FUNCTION_BLOCK SoEReadProcess EXTENDS BaseProcess
  VAR_INPUT
    value1Byte : USINT;  (* Value that has been read, if noOfBytes is 1 *)
    value2Bytes : UINT;  (* Value that has been read, if noOfBytes is 2 *)
    value4Bytes : UDINT;  (* Value that has been read, if noOfBytes is 4 *)
    adsErrorId : UINT;  (* ADS error ID *)
    sercosErrorId : UINT;  (* Sercos error ID *)
    {attribute 'OPC.UA.DA' := '1'}
    set : SoEReadProcessArgs;  (* Arguments to be set, before writing do_request TRUE *)
  END_VAR
  VAR_OUTPUT
    {attribute 'OPC.UA.DA' := '1'}
    {attribute 'OPC.UA.DA.Access' := '1'}
    get : SoEReadProcessArgs;  (* Arguments in use by the process, if do_request was accepted *)
  END_VAR

            IF do_request THEN
    do_request_result := request(
    index := set.index,
    noOfBytes := set.noOfBytes);
    do_request := FALSE;
END_IF;
SUPER^();

          

{attribute 'TcRpcEnable' := '1'}
METHOD start
  VAR_INPUT
    index : UINT;  (* SDO Index *)
    noOfBytes : UDINT;  (* Number of bytes to be read *)
  END_VAR
                  THIS^.get.index := index;
THIS^.get.noOfBytes := noOfBytes;
THIS^.statuses.busyStatus( isBusy := TRUE );
THIS^.statuses.healthStatus( isGood := TRUE );

                
END_METHOD

{attribute 'TcRpcEnable' := '1'}
METHOD request : RequestResults
  VAR_INPUT
    index : UINT;  (* SDO Index *)
    noOfBytes : UDINT;  (* Number of bytes to be read *)
  END_VAR
                  IF THIS^.statuses.enabledStatus.enabled THEN
    request := RequestResults.ACCEPTED;
    THIS^.start(
        index := index,
        noOfBytes := noOfBytes);
ELSE
    request := RequestResults.REJECTED;
END_IF;

                
END_METHOD
END_FUNCTION_BLOCK

FUNCTION_BLOCK SoEWriteProcess EXTENDS BaseProcess
  VAR_INPUT
    adsErrorId : UINT;  (* ADS error ID *)
    sercosErrorId : UINT;  (* Sercos error ID *)
    {attribute 'OPC.UA.DA' := '1'}
    set : SoEWriteProcessArgs;  (* Arguments to be set, before writing do_request TRUE *)
  END_VAR
  VAR_OUTPUT
    {attribute 'OPC.UA.DA' := '1'}
    {attribute 'OPC.UA.DA.Access' := '1'}
    get : SoEWriteProcessArgs;  (* Arguments in use by the process, if do_request was accepted *)
  END_VAR

            IF do_request THEN
    do_request_result := request(
    index := set.index,
    noOfBytes := set.noOfBytes,
    value1Byte := set.value1Byte,
    value2Bytes := set.value2Bytes,
    value4Bytes := set.value4Bytes);
    do_request := FALSE;
END_IF;
SUPER^();

          

{attribute 'TcRpcEnable' := '1'}
METHOD start
  VAR_INPUT
    index : UINT;  (* SDO Index *)
    noOfBytes : UDINT;  (* Number of bytes to be written *)
    value1Byte : USINT;  (* Value to be written if noOfBytes is 1 *)
    value2Bytes : UINT;  (* Value to be written if noOfBytes is 2 *)
    value4Bytes : UDINT;  (* Value to be written if noOfBytes is 4 *)
  END_VAR
                  THIS^.get.index := index;
THIS^.get.noOfBytes := noOfBytes;
THIS^.get.value1Byte := value1Byte;
THIS^.get.value2Bytes := value2Bytes;
THIS^.get.value4Bytes := value4Bytes;
THIS^.statuses.busyStatus( isBusy := TRUE );
THIS^.statuses.healthStatus( isGood := TRUE );

                
END_METHOD

{attribute 'TcRpcEnable' := '1'}
METHOD request : RequestResults
  VAR_INPUT
    index : UINT;  (* SDO Index *)
    noOfBytes : UDINT;  (* Number of bytes to be written *)
    value1Byte : USINT;  (* Value to be written if noOfBytes is 1 *)
    value2Bytes : UINT;  (* Value to be written if noOfBytes is 2 *)
    value4Bytes : UDINT;  (* Value to be written if noOfBytes is 4 *)
  END_VAR
                  IF THIS^.statuses.enabledStatus.enabled THEN
    request := RequestResults.ACCEPTED;
    THIS^.start(
        index := index,
        noOfBytes := noOfBytes,
        value1Byte := value1Byte,
        value2Bytes := value2Bytes,
        value4Bytes := value4Bytes);
ELSE
    request := RequestResults.REJECTED;
END_IF;

                
END_METHOD
END_FUNCTION_BLOCK

FUNCTION_BLOCK SoEResetProcess EXTENDS BaseProcess
  VAR_INPUT
    adsErrorId : UINT;  (* ADS error ID *)
    sercosErrorId : UINT;  (* Sercos error ID *)
  END_VAR

            IF do_request THEN
    do_request_result := request();
    do_request := FALSE;
END_IF;
SUPER^();

          

{attribute 'TcRpcEnable' := '1'}
METHOD start
                  THIS^.statuses.busyStatus( isBusy := TRUE );
THIS^.statuses.healthStatus( isGood := TRUE );

                
END_METHOD

{attribute 'TcRpcEnable' := '1'}
METHOD request : RequestResults
                  IF THIS^.statuses.enabledStatus.enabled THEN
    request := RequestResults.ACCEPTED;
    THIS^.start();
ELSE
    request := RequestResults.REJECTED;
END_IF;

                
END_METHOD
END_FUNCTION_BLOCK

FUNCTION_BLOCK SetBrakeProcess EXTENDS BaseProcess
  VAR_INPUT
    {attribute 'OPC.UA.DA' := '1'}
    set : SetBrakeProcessArgs;  (* Arguments to be set, before writing do_request TRUE *)
  END_VAR
  VAR_OUTPUT
    {attribute 'OPC.UA.DA' := '1'}
    {attribute 'OPC.UA.DA.Access' := '1'}
    get : SetBrakeProcessArgs;  (* Arguments in use by the process, if do_request was accepted *)
  END_VAR

            IF do_request THEN
    do_request_result := request( newState := set.newState );
    do_request := FALSE;
END_IF;
SUPER^();

          

{attribute 'TcRpcEnable' := '1'}
METHOD start
  VAR_INPUT
    newState : DriveBrakeStates;  (* Requested brake state *)
  END_VAR
                  THIS^.get.newState := newState;
THIS^.statuses.busyStatus( isBusy := TRUE );
THIS^.statuses.healthStatus( isGood := TRUE );

                
END_METHOD

{attribute 'TcRpcEnable' := '1'}
METHOD request : RequestResults
  VAR_INPUT
    newState : DriveBrakeStates;  (* Requested brake state *)
  END_VAR
                  IF THIS^.statuses.enabledStatus.enabled THEN
    request := RequestResults.ACCEPTED;
    THIS^.start( newState := newState );
ELSE
    request := RequestResults.REJECTED;
END_IF;

                
END_METHOD
END_FUNCTION_BLOCK

FUNCTION_BLOCK ChangeOperatingStateProcess EXTENDS BaseProcess
  VAR_INPUT
    {attribute 'OPC.UA.DA' := '1'}
    set : ChangeOperatingStateProcessArgs;  (* Arguments to be set, before writing do_request TRUE *)
  END_VAR
  VAR_OUTPUT
    {attribute 'OPC.UA.DA' := '1'}
    {attribute 'OPC.UA.DA.Access' := '1'}
    get : ChangeOperatingStateProcessArgs;  (* Arguments in use by the process, if do_request was accepted *)
  END_VAR

            IF do_request THEN
    do_request_result := request( state := set.state );
    do_request := FALSE;
END_IF;
SUPER^();

          

{attribute 'TcRpcEnable' := '1'}
METHOD start
  VAR_INPUT
    state : OperatingStates;  (* New operating state (e.g. AUTO, MANUAL) *)
  END_VAR
                  THIS^.get.state := state;
THIS^.statuses.busyStatus( isBusy := TRUE );
THIS^.statuses.healthStatus( isGood := TRUE );

                
END_METHOD

{attribute 'TcRpcEnable' := '1'}
METHOD request : RequestResults
  VAR_INPUT
    state : OperatingStates;  (* New operating state (e.g. AUTO, MANUAL) *)
  END_VAR
                  IF THIS^.statuses.enabledStatus.enabled THEN
    request := RequestResults.ACCEPTED;
    THIS^.start( state := state );
ELSE
    request := RequestResults.REJECTED;
END_IF;

                
END_METHOD
END_FUNCTION_BLOCK

FUNCTION_BLOCK ChangeOperatorStateProcess EXTENDS BaseProcess
  VAR_INPUT
    {attribute 'OPC.UA.DA' := '1'}
    set : ChangeOperatorStateProcessArgs;  (* Arguments to be set, before writing do_request TRUE *)
  END_VAR
  VAR_OUTPUT
    {attribute 'OPC.UA.DA' := '1'}
    {attribute 'OPC.UA.DA.Access' := '1'}
    get : ChangeOperatorStateProcessArgs;  (* Arguments in use by the process, if do_request was accepted *)
  END_VAR

            IF do_request THEN
    do_request_result := request(
    state := set.state,
    password := set.password);
    do_request := FALSE;
END_IF;
SUPER^();

          

{attribute 'TcRpcEnable' := '1'}
METHOD start
  VAR_INPUT
    state : OperatorStates;  (* New operator state (e.g. OBSERVER, TECH, ...) *)
    password : STRING;  (* Password (only sometimes required, e.g. to go from OBSERVER to TECH) *)
  END_VAR
                  THIS^.get.state := state;
THIS^.get.password := password;
THIS^.statuses.busyStatus( isBusy := TRUE );
THIS^.statuses.healthStatus( isGood := TRUE );

                
END_METHOD

{attribute 'TcRpcEnable' := '1'}
METHOD request : RequestResults
  VAR_INPUT
    state : OperatorStates;  (* New operator state (e.g. OBSERVER, TECH, ...) *)
    password : STRING;  (* Password (only sometimes required, e.g. to go from OBSERVER to TECH) *)
  END_VAR
                  IF THIS^.statuses.enabledStatus.enabled THEN
    request := RequestResults.ACCEPTED;
    THIS^.start(
        state := state,
        password := password);
ELSE
    request := RequestResults.REJECTED;
END_IF;

                
END_METHOD
END_FUNCTION_BLOCK

FUNCTION_BLOCK ChangeOperatingModeStateProcess EXTENDS BaseProcess
  VAR_INPUT
    {attribute 'OPC.UA.DA' := '1'}
    set : ChangeOperatingModeStateProcessArgs;  (* Arguments to be set, before writing do_request TRUE *)
  END_VAR
  VAR_OUTPUT
    {attribute 'OPC.UA.DA' := '1'}
    {attribute 'OPC.UA.DA.Access' := '1'}
    get : ChangeOperatingModeStateProcessArgs;  (* Arguments in use by the process, if do_request was accepted *)
  END_VAR

            IF do_request THEN
    do_request_result := request( state := set.state );
    do_request := FALSE;
END_IF;
SUPER^();

          

{attribute 'TcRpcEnable' := '1'}
METHOD start
  VAR_INPUT
    state : OperatingModeStates;  (* New operating state (e.g. LOCAL, REMOTE) *)
  END_VAR
                  THIS^.get.state := state;
THIS^.statuses.busyStatus( isBusy := TRUE );
THIS^.statuses.healthStatus( isGood := TRUE );

                
END_METHOD

{attribute 'TcRpcEnable' := '1'}
METHOD request : RequestResults
  VAR_INPUT
    state : OperatingModeStates;  (* New operating state (e.g. LOCAL, REMOTE) *)
  END_VAR
                  IF THIS^.statuses.enabledStatus.enabled THEN
    request := RequestResults.ACCEPTED;
    THIS^.start( state := state );
ELSE
    request := RequestResults.REJECTED;
END_IF;

                
END_METHOD
END_FUNCTION_BLOCK

FUNCTION_BLOCK ReadXmlProcess EXTENDS BaseXmlDataSrvProcess
  VAR_INPUT
    {attribute 'OPC.UA.DA' := '1'}
    set : ReadXmlProcessArgs;  (* Arguments to be set, before writing do_request TRUE *)
  END_VAR
  VAR_OUTPUT
    {attribute 'OPC.UA.DA' := '1'}
    {attribute 'OPC.UA.DA.Access' := '1'}
    get : ReadXmlProcessArgs;  (* Arguments in use by the process, if do_request was accepted *)
  END_VAR

            IF do_request THEN
    do_request_result := request( filePath := set.filePath );
    do_request := FALSE;
END_IF;
SUPER^();

          

{attribute 'TcRpcEnable' := '1'}
METHOD start
  VAR_INPUT
    filePath : STRING;  (* Full path of the filename to read *)
  END_VAR
                  THIS^.get.filePath := filePath;
THIS^.statuses.busyStatus( isBusy := TRUE );
THIS^.statuses.healthStatus( isGood := TRUE );

                
END_METHOD

{attribute 'TcRpcEnable' := '1'}
METHOD request : RequestResults
  VAR_INPUT
    filePath : STRING;  (* Full path of the filename to read *)
  END_VAR
                  IF THIS^.statuses.enabledStatus.enabled THEN
    request := RequestResults.ACCEPTED;
    THIS^.start( filePath := filePath );
ELSE
    request := RequestResults.REJECTED;
END_IF;

                
END_METHOD
END_FUNCTION_BLOCK

FUNCTION_BLOCK WriteXmlProcess EXTENDS BaseXmlDataSrvProcess
  VAR_INPUT
    {attribute 'OPC.UA.DA' := '1'}
    set : WriteXmlProcessArgs;  (* Arguments to be set, before writing do_request TRUE *)
  END_VAR
  VAR_OUTPUT
    {attribute 'OPC.UA.DA' := '1'}
    {attribute 'OPC.UA.DA.Access' := '1'}
    get : WriteXmlProcessArgs;  (* Arguments in use by the process, if do_request was accepted *)
  END_VAR

            IF do_request THEN
    do_request_result := request( filePath := set.filePath );
    do_request := FALSE;
END_IF;
SUPER^();

          

{attribute 'TcRpcEnable' := '1'}
METHOD start
  VAR_INPUT
    filePath : STRING;  (* Full path of the filename to write *)
  END_VAR
                  THIS^.get.filePath := filePath;
THIS^.statuses.busyStatus( isBusy := TRUE );
THIS^.statuses.healthStatus( isGood := TRUE );

                
END_METHOD

{attribute 'TcRpcEnable' := '1'}
METHOD request : RequestResults
  VAR_INPUT
    filePath : STRING;  (* Full path of the filename to write *)
  END_VAR
                  IF THIS^.statuses.enabledStatus.enabled THEN
    request := RequestResults.ACCEPTED;
    THIS^.start( filePath := filePath );
ELSE
    request := RequestResults.REJECTED;
END_IF;

                
END_METHOD
END_FUNCTION_BLOCK

FUNCTION_BLOCK ActivateProcess EXTENDS BaseProcess
  VAR
    {attribute 'OPC.UA.DA' := '0'}
    testVar : BOOL;  (* At least 1 variable needed because subclass members of an empty class are not exposed by OPC UA (TwinCAT bug!) *)
  END_VAR

            IF do_request THEN
    do_request_result := request();
    do_request := FALSE;
END_IF;
SUPER^();

          

{attribute 'TcRpcEnable' := '1'}
METHOD start
                  THIS^.statuses.busyStatus( isBusy := TRUE );
THIS^.statuses.healthStatus( isGood := TRUE );

                
END_METHOD

{attribute 'TcRpcEnable' := '1'}
METHOD request : RequestResults
                  IF THIS^.statuses.enabledStatus.enabled THEN
    request := RequestResults.ACCEPTED;
    THIS^.start();
ELSE
    request := RequestResults.REJECTED;
END_IF;

                
END_METHOD
END_FUNCTION_BLOCK

FUNCTION_BLOCK ModbusRTUBusReadCoilProcess EXTENDS BaseProcess
  VAR_INPUT
    value : BOOL;  (* Value of the coil *)
    errorId : INT;  (* Error Id. Modbus error code *)
    {attribute 'OPC.UA.DA' := '1'}
    set : ModbusRTUBusReadCoilProcessArgs;  (* Arguments to be set, before writing do_request TRUE *)
  END_VAR
  VAR_OUTPUT
    {attribute 'OPC.UA.DA' := '1'}
    {attribute 'OPC.UA.DA.Access' := '1'}
    get : ModbusRTUBusReadCoilProcessArgs;  (* Arguments in use by the process, if do_request was accepted *)
  END_VAR

            IF do_request THEN
    do_request_result := request(
    unitID := set.unitID,
    address := set.address);
    do_request := FALSE;
END_IF;
SUPER^();

          

{attribute 'TcRpcEnable' := '1'}
METHOD start
  VAR_INPUT
    unitID : USINT;  (* Modbus station address (1..247) *)
    address : UINT;  (* Modbus data address *)
  END_VAR
                  THIS^.get.unitID := unitID;
THIS^.get.address := address;
THIS^.statuses.busyStatus( isBusy := TRUE );
THIS^.statuses.healthStatus( isGood := TRUE );

                
END_METHOD

{attribute 'TcRpcEnable' := '1'}
METHOD request : RequestResults
  VAR_INPUT
    unitID : USINT;  (* Modbus station address (1..247) *)
    address : UINT;  (* Modbus data address *)
  END_VAR
                  IF THIS^.statuses.enabledStatus.enabled THEN
    request := RequestResults.ACCEPTED;
    THIS^.start(
        unitID := unitID,
        address := address);
ELSE
    request := RequestResults.REJECTED;
END_IF;

                
END_METHOD
END_FUNCTION_BLOCK

FUNCTION_BLOCK ModbusRTUBusWriteCoilProcess EXTENDS BaseProcess
  VAR_INPUT
    errorId : INT;  (* Error Id. Modbus error code *)
    {attribute 'OPC.UA.DA' := '1'}
    set : ModbusRTUBusWriteCoilProcessArgs;  (* Arguments to be set, before writing do_request TRUE *)
  END_VAR
  VAR_OUTPUT
    {attribute 'OPC.UA.DA' := '1'}
    {attribute 'OPC.UA.DA.Access' := '1'}
    get : ModbusRTUBusWriteCoilProcessArgs;  (* Arguments in use by the process, if do_request was accepted *)
  END_VAR

            IF do_request THEN
    do_request_result := request(
    unitID := set.unitID,
    address := set.address,
    value := set.value);
    do_request := FALSE;
END_IF;
SUPER^();

          

{attribute 'TcRpcEnable' := '1'}
METHOD start
  VAR_INPUT
    unitID : USINT;  (* Modbus station address (1..247) *)
    address : UINT;  (* Modbus data address *)
    value : BOOL;  (* Value to write on the coil *)
  END_VAR
                  THIS^.get.unitID := unitID;
THIS^.get.address := address;
THIS^.get.value := value;
THIS^.statuses.busyStatus( isBusy := TRUE );
THIS^.statuses.healthStatus( isGood := TRUE );

                
END_METHOD

{attribute 'TcRpcEnable' := '1'}
METHOD request : RequestResults
  VAR_INPUT
    unitID : USINT;  (* Modbus station address (1..247) *)
    address : UINT;  (* Modbus data address *)
    value : BOOL;  (* Value to write on the coil *)
  END_VAR
                  IF THIS^.statuses.enabledStatus.enabled THEN
    request := RequestResults.ACCEPTED;
    THIS^.start(
        unitID := unitID,
        address := address,
        value := value);
ELSE
    request := RequestResults.REJECTED;
END_IF;

                
END_METHOD
END_FUNCTION_BLOCK

FUNCTION_BLOCK ModbusRTUBusReadRegisterProcess EXTENDS BaseProcess
  VAR_INPUT
    value : INT;  (* Value of the register *)
    errorId : INT;  (* Error Id. Modbus error code *)
    {attribute 'OPC.UA.DA' := '1'}
    set : ModbusRTUBusReadRegisterProcessArgs;  (* Arguments to be set, before writing do_request TRUE *)
  END_VAR
  VAR_OUTPUT
    {attribute 'OPC.UA.DA' := '1'}
    {attribute 'OPC.UA.DA.Access' := '1'}
    get : ModbusRTUBusReadRegisterProcessArgs;  (* Arguments in use by the process, if do_request was accepted *)
  END_VAR

            IF do_request THEN
    do_request_result := request(
    unitID := set.unitID,
    address := set.address);
    do_request := FALSE;
END_IF;
SUPER^();

          

{attribute 'TcRpcEnable' := '1'}
METHOD start
  VAR_INPUT
    unitID : USINT;  (* Modbus station address (1..247) *)
    address : UINT;  (* Modbus data address *)
  END_VAR
                  THIS^.get.unitID := unitID;
THIS^.get.address := address;
THIS^.statuses.busyStatus( isBusy := TRUE );
THIS^.statuses.healthStatus( isGood := TRUE );

                
END_METHOD

{attribute 'TcRpcEnable' := '1'}
METHOD request : RequestResults
  VAR_INPUT
    unitID : USINT;  (* Modbus station address (1..247) *)
    address : UINT;  (* Modbus data address *)
  END_VAR
                  IF THIS^.statuses.enabledStatus.enabled THEN
    request := RequestResults.ACCEPTED;
    THIS^.start(
        unitID := unitID,
        address := address);
ELSE
    request := RequestResults.REJECTED;
END_IF;

                
END_METHOD
END_FUNCTION_BLOCK

FUNCTION_BLOCK ModbusRTUBusWriteRegisterProcess EXTENDS BaseProcess
  VAR_INPUT
    errorId : INT;  (* Error Id. Modbus error code *)
    {attribute 'OPC.UA.DA' := '1'}
    set : ModbusRTUBusWriteRegisterProcessArgs;  (* Arguments to be set, before writing do_request TRUE *)
  END_VAR
  VAR_OUTPUT
    {attribute 'OPC.UA.DA' := '1'}
    {attribute 'OPC.UA.DA.Access' := '1'}
    get : ModbusRTUBusWriteRegisterProcessArgs;  (* Arguments in use by the process, if do_request was accepted *)
  END_VAR

            IF do_request THEN
    do_request_result := request(
    unitID := set.unitID,
    address := set.address,
    value := set.value);
    do_request := FALSE;
END_IF;
SUPER^();

          

{attribute 'TcRpcEnable' := '1'}
METHOD start
  VAR_INPUT
    unitID : USINT;  (* Modbus station address (1..247) *)
    address : UINT;  (* Modbus data address *)
    value : INT;  (* Value to write on the register *)
  END_VAR
                  THIS^.get.unitID := unitID;
THIS^.get.address := address;
THIS^.get.value := value;
THIS^.statuses.busyStatus( isBusy := TRUE );
THIS^.statuses.healthStatus( isGood := TRUE );

                
END_METHOD

{attribute 'TcRpcEnable' := '1'}
METHOD request : RequestResults
  VAR_INPUT
    unitID : USINT;  (* Modbus station address (1..247) *)
    address : UINT;  (* Modbus data address *)
    value : INT;  (* Value to write on the register *)
  END_VAR
                  IF THIS^.statuses.enabledStatus.enabled THEN
    request := RequestResults.ACCEPTED;
    THIS^.start(
        unitID := unitID,
        address := address,
        value := value);
ELSE
    request := RequestResults.REJECTED;
END_IF;

                
END_METHOD
END_FUNCTION_BLOCK

FUNCTION_BLOCK ModbusRTUBusDiagnosticsProcess EXTENDS BaseProcess
  VAR_INPUT
    value : INT;  (* Value of the register *)
    errorId : INT;  (* Error Id. Modbus error code *)
    {attribute 'OPC.UA.DA' := '1'}
    set : ModbusRTUBusDiagnosticsProcessArgs;  (* Arguments to be set, before writing do_request TRUE *)
  END_VAR
  VAR_OUTPUT
    {attribute 'OPC.UA.DA' := '1'}
    {attribute 'OPC.UA.DA.Access' := '1'}
    get : ModbusRTUBusDiagnosticsProcessArgs;  (* Arguments in use by the process, if do_request was accepted *)
  END_VAR

            IF do_request THEN
    do_request_result := request(
    unitID := set.unitID,
    subFunction := set.subFunction,
    subData := set.subData);
    do_request := FALSE;
END_IF;
SUPER^();

          

{attribute 'TcRpcEnable' := '1'}
METHOD start
  VAR_INPUT
    unitID : USINT;  (* Modbus station address (1..247) *)
    subFunction : UINT;  (* Modbus subFunction code *)
    subData : INT;  (* Modbus data for subFunction *)
  END_VAR
                  THIS^.get.unitID := unitID;
THIS^.get.subFunction := subFunction;
THIS^.get.subData := subData;
THIS^.statuses.busyStatus( isBusy := TRUE );
THIS^.statuses.healthStatus( isGood := TRUE );

                
END_METHOD

{attribute 'TcRpcEnable' := '1'}
METHOD request : RequestResults
  VAR_INPUT
    unitID : USINT;  (* Modbus station address (1..247) *)
    subFunction : UINT;  (* Modbus subFunction code *)
    subData : INT;  (* Modbus data for subFunction *)
  END_VAR
                  IF THIS^.statuses.enabledStatus.enabled THEN
    request := RequestResults.ACCEPTED;
    THIS^.start(
        unitID := unitID,
        subFunction := subFunction,
        subData := subData);
ELSE
    request := RequestResults.REJECTED;
END_IF;

                
END_METHOD
END_FUNCTION_BLOCK
